// TIA Portal V20 export
FUNCTION "V100" : Void   // FC3, FBD
{ S7_Optimized_Access := 'TRUE' }
// stored: SetENOAutomatically false
   VAR_TEMP
      Temp : "DigVal";
      Temp_1 : "DigVal";
      State : "Service_States";
   END_VAR
BEGIN

REGION Network 1: Channel input
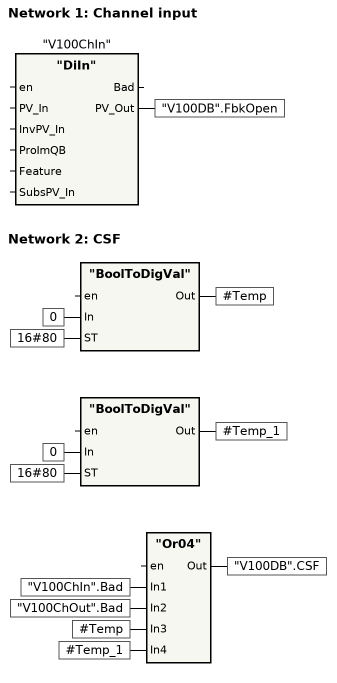
   "V100ChIn"(PV_Out => "V100DB".FbkOpen);   // "DiIn"
END_REGION

REGION Network 2: CSF
   "BoolToDigVal"(In := 0, ST := 16#80, Out => #Temp);
   "BoolToDigVal"(In := 0, ST := 16#80, Out => #Temp_1);
   "Or04"(In1 := "V100ChIn".Bad, In2 := "V100ChOut".Bad, In3 := #Temp, In4 := #Temp_1, Out => "V100DB".CSF);
END_REGION

REGION Network 3: VlvAn Intlock
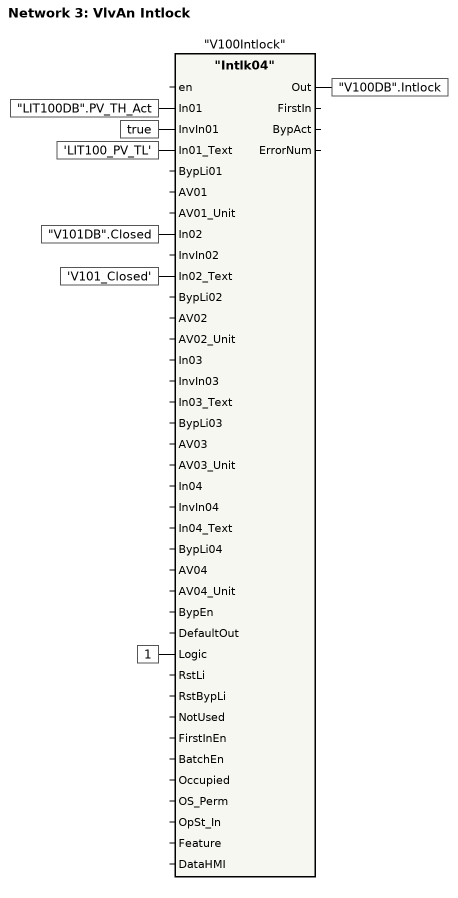
   "V100Intlock"(In01 := "LIT100DB".PV_TH_Act,   // "Intlk04"
                 InvIn01 := true,
                 In01_Text := 'LIT100_PV_TL',
                 In02 := "V101DB".Closed,
                 In02_Text := 'V101_Closed',
                 Logic := 1,
                 Out => "V100DB".Intlock);
END_REGION

REGION Network 4: VlvAnL
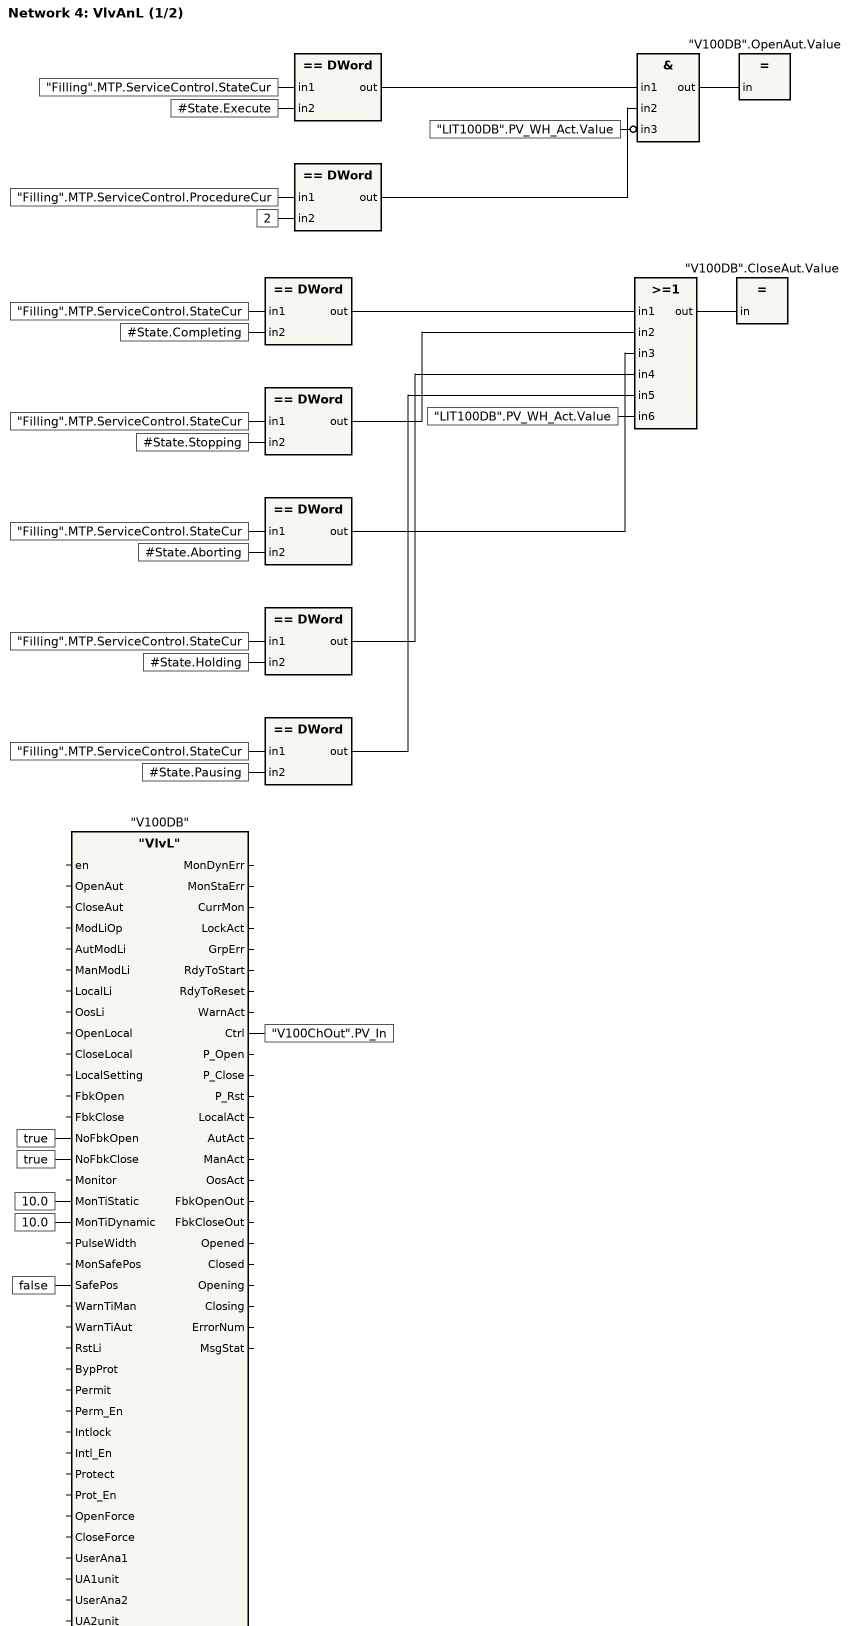
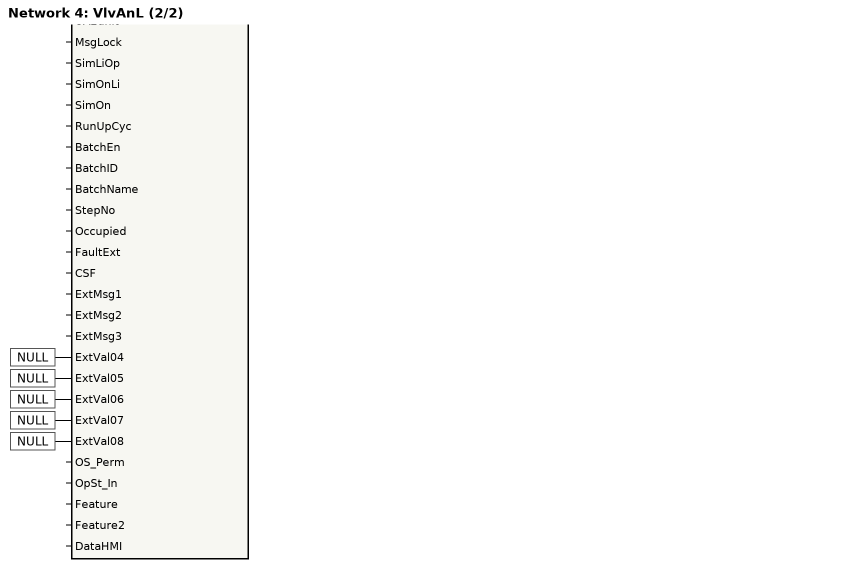
   "V100DB".OpenAut.Value := ("Filling".MTP.ServiceControl.StateCur = #State.Execute) AND ("Filling".MTP.ServiceControl.ProcedureCur = 2) AND NOT "LIT100DB".PV_WH_Act.Value;
   "V100DB".CloseAut.Value := ("Filling".MTP.ServiceControl.StateCur = #State.Completing) OR ("Filling".MTP.ServiceControl.StateCur = #State.Stopping) OR ("Filling".MTP.ServiceControl.StateCur = #State.Aborting) OR ("Filling".MTP.ServiceControl.StateCur = #State.Holding) OR ("Filling".MTP.ServiceControl.StateCur = #State.Pausing) OR "LIT100DB".PV_WH_Act.Value;
   "V100DB"(NoFbkOpen := true,   // "VlvL"
            NoFbkClose := true,
            MonTiStatic := 10.0,
            MonTiDynamic := 10.0,
            SafePos := false,
            ExtVal04 := NULL,
            ExtVal05 := NULL,
            ExtVal06 := NULL,
            ExtVal07 := NULL,
            ExtVal08 := NULL,
            Ctrl => "V100ChOut".PV_In);
END_REGION

REGION Network 5: MTP
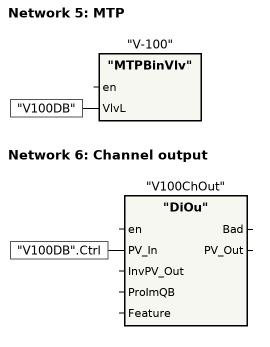
   "V-100"(VlvL := "V100DB");   // "MTPBinVlv"
END_REGION

REGION Network 6: Channel output
   "V100ChOut"(PV_In := "V100DB".Ctrl);   // "DiOu"
END_REGION
END_FUNCTION
